FUNCTION F_SAFETY_StatusFB_TO_EDM : ST_SAFETY_FBEDM
VAR_INPUT
	stFBStatus						: ST_SAFETY_FBStatus; 	(* Struktura ogolna *)
END_VAR

F_SAFETY_StatusFB_TO_EDM.uStatus.stStatusWords	:= stFBStatus;									(* Przepisanie *)
F_SAFETY_StatusFB_TO_EDM.eState 				:= stFBStatus.BState;							(* Ustawienie enum *)
F_SAFETY_StatusFB_TO_EDM.bGeneralError			:= stFBStatus.wDiagnosis <> 0;					(* General Error *)

END_FUNCTION

(* stored: Version 1.1.0.1, ProductVersion 3.1.4022.12
   POU F_SAFETY_StatusFB_TO_EDM: Id {797010e5-f260-47ec-a939-98141bb65bc0}, SpecialFunc None *)
